TYPE aS_DBField :
STRUCT
	Id: LINT;
	Sync: BOOL;
	Timestamp: DT;
	FurTemp: REAL;
	FurInper: REAL;
	LphTemp: REAL;
	LphPress: REAL;
	LphInpress: REAL;
	LphInflow: REAL;
	DeaTemp: REAL;
	DeaPress: REAL;
	HphTemp: REAL;
	HphPress: REAL;
	HphInpress: REAL;
	HphInflow: REAL;
	BoiTemp: REAL;
	BoiPress: REAL;
	ConTemp: REAL;
	ConInflow: REAL;
	TurHtemp: REAL;
	TurItemp: REAL;
	TurLtemp: REAL;
	TurHpress: REAL;
	TurIpress: REAL;
	TurLpress: REAL;
	TurSpeed: REAL;
END_STRUCT
END_TYPE

(* stored: Version 1.1.0.1, ProductVersion 3.1.4024.4
   DUT aS_DBField: Id {1650d890-ddeb-4e8e-9353-f87e78cac51e} *)
